PROGRAM Axis01_Interlock
VAR
//System_Bit
	Always_ON	:	BOOL	:=TRUE	;//상시 ON 
	Always_OFF	:	BOOL	:=FALSE	;//상시 OFF
END_VAR

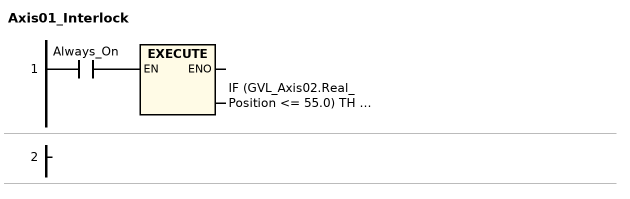
// NETWORK 1
IF Always_On THEN
    IF (GVL_Axis02.Real_Position <= 55.0) THEN
    	GVL_Axis01.Interlock := TRUE;
    END_IF
    IF (GVL_Axis02.Real_Position >= 55.0) THEN
    	IF GVL_Axis01.Selected_Position_Data
    > 0.0 THEN
    		GVL_Axis01.Interlock := True;
    	END_IF
    END_IF
END_IF

// NETWORK 2

END_PROGRAM

(* stored: Version 1.1.0.1, ProductVersion 3.1.4024.15
   POU Axis01_Interlock: Id {1a2871bf-aa4d-4f83-9338-80c18a49dc56}, SpecialFunc None *)
